Yaskawa INFORM job: SKRZYNIA_4040_-90_STOPNI_20BR.JBI

/JOB
//NAME SKRZYNIA_4040_-90_STOPNI_20BR
///FOLDERNAME 02-SKRZYNIE_JOBS
//POS
///NPOS 307,307,0,21,0,0
///TOOL 0
///POSTYPE PULSE
///PULSE
C00000=0,-52280,40443,0,6876,0
C00001=-82314,-24956,17040,-59626,-27382,-6248
C00002=-93910,-8625,17040,-59626,-43355,-6248
C00003=-98846,-1061,-42166,-80308,-57081,16120
C00004=-100452,6057,-48127,-85711,-56704,21322
C00005=-95817,31791,-34187,-84788,-63710,26674
C00006=-95573,33077,-33257,-84645,-64023,26851
C00007=-94315,33778,-32137,-85160,-63467,26714
C00008=-95573,33077,-33257,-84645,-64023,26851
C00009=-94948,31301,-36075,-85235,-63717,27152
C00010=-95573,33077,-33257,-84645,-64023,26851
C00011=-95263,33142,-33256,-84677,-63995,26850
C00012=-95263,33142,-33256,-84677,-63995,26850
C00013=-94230,33719,-32331,-85099,-63538,26735
C00014=-95263,33142,-33256,-84677,-63995,26850
C00015=-94794,31816,-35365,-85120,-63763,27076
C00016=-95263,33142,-33256,-84677,-63995,26850
C00017=-95260,33144,-33256,-84678,-63995,26850
C00018=-95260,33144,-33256,-84678,-63995,26850
C00019=-94260,33701,-32361,-85086,-63552,26738
C00020=-95738,35616,-30155,-83417,-65710,26451
C00021=-94835,31943,-35167,-85080,-63786,27056
C00022=-95260,33144,-33256,-84678,-63995,26850
C00023=-95258,25631,32269,-66559,-75499,2416
C00024=-95258,25631,32269,-66559,-75499,2416
C00025=-94256,26435,33444,-66420,-74940,2208
C00026=-95258,25631,32269,-66559,-75499,2416
C00027=-94857,24030,29962,-66606,-75105,2539
C00028=-95258,25631,32269,-66559,-75499,2416
C00029=-98811,21047,-15512,-99242,-81394,20987
C00030=-98811,21047,-15512,-99242,-81394,20987
C00031=-97856,21592,-14760,-99539,-80803,20995
C00032=-98811,21047,-15512,-99242,-81394,20987
C00033=-98487,19855,-17143,-99373,-81250,21110
C00034=-98811,21047,-15512,-99242,-81394,20987
C00035=-100395,5963,-6492,-101051,-69866,13942
C00036=-97697,-21147,-29798,-104770,-52931,14344
C00037=-81691,-45027,-49520,-104186,-37412,14105
C00038=-48287,-44591,-17414,-16172,-14532,-25809
C00039=-85348,-13130,13838,-41209,-47455,-8220
C00040=-97998,22495,32685,-69647,-75009,8900
C00041=-98284,29564,37770,-71835,-80250,10571
C00042=-100615,26523,30326,-83718,-79542,3747
C00043=-99528,26746,30653,-83688,-78804,3698
C00044=-98609,27389,31597,-83640,-78189,3601
C00045=-99528,26746,30653,-83688,-78804,3698
C00046=-99278,25562,28929,-83734,-78615,3833
C00047=-99528,26746,30653,-83688,-78804,3698
C00048=-97827,29852,38067,-72347,-79830,10157
C00049=-97362,30289,38867,-71738,-79704,10396
C00050=-96447,31020,39967,-71637,-79179,10220
C00051=-97362,30289,38867,-71738,-79704,10396
C00052=-97069,28896,36765,-71776,-79401,10550
C00053=-97362,30289,38867,-71738,-79704,10396
C00054=-99687,30516,41738,-96594,-77984,-2813
C00055=-99279,34023,49568,-96204,-78485,-4167
C00056=-98297,34881,50932,-96068,-77785,-4257
C00057=-99279,34023,49568,-96204,-78485,-4167
C00058=-98948,32155,46632,-96284,-78364,-3863
C00059=-99279,34023,49568,-96204,-78485,-4167
C00060=-100799,20404,12473,-99797,-78179,2590
C00061=-99814,-4938,-36996,-116444,-71342,12229
C00062=-82620,-30758,-83593,-142203,-62652,21635
C00063=-79591,-62427,-80212,-133576,-39445,13545
C00064=-61872,-66272,-83954,-148251,-32298,21081
C00065=-61872,-49557,-32264,-110357,-15428,1928
C00066=-71091,-37860,2722,-34648,-42002,-27792
C00067=-94097,-13222,20403,-45591,-54273,-19204
C00068=-97363,-23488,-17584,-60839,-44712,-9276
C00069=-98197,-8670,-25604,-81540,-55001,4479
C00070=-99236,18416,3235,-80713,-73731,6125
C00071=-98716,22747,8680,-80557,-75862,6048
C00072=-97982,23215,9333,-80619,-75386,5974
C00073=-98716,22747,8680,-80557,-75862,6048
C00074=-98409,21490,6932,-80649,-75627,6156
C00075=-98716,22747,8680,-80557,-75862,6048
C00076=-94729,-288,3800,-87543,-55904,1533
C00077=-77861,-26606,-19905,-76223,-21443,-3330
C00078=-46440,-50562,-32626,1826,-13880,-39178
C00079=-46440,-50562,-32626,1826,-13880,-39178
///LIMIT ON
C00080=-38692,-65390,10180,-18335,3144,1955
///LIMIT OFF
C00081=0,-52280,40443,0,6876,0
C00082=0,-52280,40443,0,6876,0
C00083=0,-43112,23163,32261,-40956,29092
C00084=-48283,-21883,28214,-25170,-26491,48363
C00085=-46664,-3144,58041,-18842,-32105,45325
C00086=-50347,-18571,12268,-49104,-16423,60029
C00087=-50509,-19000,10610,-51503,-15997,61182
C00088=-52966,-16930,12240,-56194,-17032,63176
C00089=-51879,-15912,13067,-55265,-16346,62852
C00090=-52154,-16175,12851,-55507,-16521,62938
C00091=-53227,-15612,13314,-57215,-17042,63646
C00092=-52966,-16930,12240,-56194,-17032,63176
C00093=-50703,-18403,11066,-52155,-16024,61477
C00094=-52780,-17619,11680,-55562,-17015,62889
C00095=-51306,-16241,12790,-54268,-16084,62435
C00096=-51660,-16583,12512,-54593,-16308,62551
C00097=-53327,-15718,13220,-57282,-17114,63667
C00098=-52780,-17619,11680,-55562,-17015,62889
C00099=-50704,-18401,11069,-52157,-16021,61478
C00100=-53191,-17342,11901,-56260,-17204,63181
C00101=-51773,-16022,12969,-55050,-16305,62760
C00102=-52146,-16378,12679,-55379,-16540,62876
C00103=-53214,-15820,13135,-57085,-17059,63584
C00104=-53002,-17172,12037,-56105,-17083,63128
C00105=-51005,-17995,11387,-52847,-16122,61778
C00106=-52654,-17319,11922,-55560,-16911,62904
C00107=-51372,-16113,12897,-54432,-16099,62508
C00108=-51648,-16379,12679,-54684,-16273,62598
C00109=-52952,-15703,13233,-56807,-16903,63480
C00110=-53323,-17134,12070,-56539,-17248,63304
C00111=-52826,-20105,4812,-63938,-15678,66983
C00112=-52298,-19620,5183,-63681,-15322,66914
C00113=-51076,-18450,6096,-63049,-14499,66733
C00114=-51419,-18785,5831,-63233,-14731,66786
C00115=-52680,-18133,6347,-65138,-15424,67581
C00116=-52924,-19431,7025,-60935,-16175,65505
C00117=-51752,-18759,10786,-53484,-16613,62002
C00118=-52244,-17884,11471,-54682,-16766,62529
C00119=-50303,-16031,12961,-52880,-15542,61887
C00120=-50741,-16464,12607,-53310,-15818,62044
C00121=-52416,-15612,13306,-56135,-16617,63223
C00122=-51898,-18011,11369,-54129,-16600,62301
C00123=-50945,-18019,11363,-52741,-16103,61737
C00124=-51347,-17395,11856,-53690,-16237,62152
C00125=-49990,-16073,12923,-52376,-15383,61677
C00126=-50384,-16465,12603,-52769,-15629,61822
C00127=-52066,-15616,13298,-55654,-16423,63028
C00128=-51792,-17610,11685,-54205,-16494,62350
C00129=-50945,-18019,11363,-52741,-16103,61737
C00130=-50845,-17493,11778,-52895,-15987,61824
C00131=-49521,-16191,12826,-51571,-15155,61341
C00132=-49894,-16567,12520,-51958,-15389,61484
C00133=-51728,-15654,13268,-55171,-16246,62832
C00134=-51082,-17431,11827,-53280,-16102,61986
C00135=-50028,-23690,-6096,-22921,-31075,54538
C00136=-50346,-22995,-5584,-23393,-31002,54768
C00137=-48843,-21430,-4410,-21901,-30270,54078
C00138=-49178,-21788,-4683,-22239,-30433,54235
C00139=-50538,-21100,-4158,-23908,-30654,55032
C00140=-50252,-22811,-5450,-23315,-30936,54734
C00141=-49763,-24818,-32918,-23163,-28604,59699
C00142=-49144,-24298,-32242,-22455,-28505,59304
C00143=-47766,-22458,-30816,-21237,-27774,58615
C00144=-48099,-22913,-31171,-21534,-27949,58786
C00145=-49602,-21997,-30448,-23301,-28174,59772
C00146=-49259,-23869,-32392,-22880,-28141,59533
C00147=-50713,-12366,-58367,-41124,-17813,74400
C00148=-50097,-11438,-57505,-40749,-17495,74109
C00149=-49105,-9842,-55994,-40096,-16991,73614
C00150=-49355,-10250,-56383,-40269,-17116,73742
C00151=-50506,-9357,-55529,-41571,-17503,74586
C00152=-49771,-10920,-57018,-40545,-17327,73951
C00153=-46548,-30139,-39639,-20061,-27197,57955
C00154=-48797,-26670,-6576,-20404,-32539,53259
C00155=-45389,-28224,4312,-35967,-15579,54278
C00156=-40154,-51179,-915,-24203,-8234,36524
C00157=0,-52280,40443,0,6876,0
C00158=0,-52280,40443,0,6876,0
C00159=5366,-38499,37552,-33963,-10211,16191
C00160=0,-52280,40443,0,6876,0
C00161=-82314,-24956,17040,-59626,-27382,-6248
C00162=-93910,-8625,17040,-59626,-43355,-6248
C00163=-98846,-1061,-42166,-80308,-57081,16120
C00164=-100452,6057,-48127,-85711,-56704,21322
C00165=-95564,34698,-34234,-85516,-63941,27819
C00166=-94021,36658,-30981,-84167,-64832,27454
C00167=-93851,36773,-30815,-84181,-64812,27439
C00168=-95564,34698,-34234,-85516,-63941,27819
C00169=-96930,32282,-32252,-82595,-65816,26305
C00170=-93901,32995,-31122,-83953,-64436,26132
C00171=-93891,32978,-31150,-83961,-64431,26134
C00172=-96930,32282,-32252,-82595,-65816,26305
C00173=-97719,-4194,-31542,-76086,-54596,10626
C00174=-88377,-34186,-45291,-67238,-52212,2442
C00175=-73560,-62084,7826,-28695,-34737,-3666
C00176=0,-36700,24612,42871,-31823,33862
C00177=-44403,-30110,7154,-24155,-23805,45557
C00178=-51570,-19542,10947,-41619,-21811,53396
C00179=-51570,-17239,16856,-38066,-23574,51584
C00180=-55052,-13712,19754,-43494,-24529,53873
C00181=-55307,-12713,21787,-42848,-25102,53500
C00182=-40431,-28773,9158,-17648,-23273,42875
C00183=0,-36700,24612,42871,-31823,33862
C00184=0,-52280,40443,0,6876,0
C00185=0,-52280,40443,0,6876,0
C00186=-73560,-62084,7826,-28695,-34737,-3666
C00187=-88377,-34186,-45291,-67238,-52212,2442
C00188=-99860,-8392,-35780,-75647,-56000,10650
C00189=-100432,21324,12575,-83706,-77956,7498
C00190=-100432,21324,12575,-83706,-77956,7498
C00191=-97477,24790,17443,-83584,-77881,7143
C00192=-97548,25214,18044,-83537,-78171,7107
C00193=-100432,21324,12575,-83706,-77956,7498
C00194=-100473,21504,12824,-83696,-77986,7482
C00195=-97708,25565,18549,-83502,-78342,7077
C00196=-97720,26100,19317,-83456,-78605,7025
C00197=-100432,21324,12575,-83706,-77956,7498
C00198=-99336,18440,8642,-84276,-74234,7647
C00199=-97907,25479,18429,-83510,-78268,7080
C00200=-97774,25771,18838,-83486,-78362,7054
C00201=-99336,18440,8642,-84276,-74234,7647
C00202=-88887,-29565,-44699,-91336,-36715,8429
C00203=-85230,-48302,-58733,-86716,-36654,5475
C00204=-60204,-59872,-73451,-117647,-17639,18840
C00205=-57189,-26834,-7130,-38780,-31731,51561
C00206=-55949,-20676,-3191,-39588,-29733,52121
C00207=-55884,-28531,-46032,-64057,-20842,63703
C00208=-57189,-26834,-7130,-38780,-31731,51561
C00209=-41180,-61187,4729,-17280,-8498,23442
C00210=0,-52280,40443,0,6876,0
C00211=0,-52280,40443,0,6876,0
C00212=-43180,-50572,-20637,-6552,-29302,-38834
C00213=-79425,-37128,-15462,-51820,-35721,-18807
C00214=-93702,-21743,-5664,-65079,-41536,-12324
C00215=-95468,-3718,3432,-57810,-54196,-8058
C00216=-98195,18244,29331,-65465,-72367,-4307
C00217=-96728,36447,56610,-70336,-82085,-4645
C00218=-96821,31985,42520,-71106,-80277,-1800
C00219=-99571,23446,29328,-71481,-76214,-993
C00220=-98368,-15155,-15320,-68503,-52006,-4003
C00221=-90196,-30440,-22000,-63685,-45526,-9297
C00222=-44920,-50063,-20090,-8739,-29356,-37564
C00223=-50917,-40459,4132,-34421,-18173,42391
C00224=-54964,-26842,8528,-44141,-23181,52038
C00225=-51719,-20944,8196,-48593,-18539,54728
C00226=-53338,-16066,12564,-52314,-18938,56375
C00227=-53668,-14237,17353,-48629,-20286,54493
C00228=-18010,-41727,-5437,24633,-20435,23511
C00229=-41180,-61187,4729,-17280,-8498,23442
C00230=0,-52280,40443,0,6876,0
C00231=0,-52280,40443,0,6876,0
///LIMIT ON
C00232=-37721,-67612,11381,-1325,-438,-7850
///LIMIT OFF
C00233=-43180,-50572,-20637,-6552,-29302,-38834
C00234=-79425,-37128,-15462,-51820,-35721,-18807
C00235=-92377,-33385,-41303,-83059,-36844,-1354
C00236=-98043,-4314,-16897,-86107,-58749,2387
C00237=-99186,-1007,-13605,-90357,-63007,3800
C00238=-99448,23410,16807,-87478,-77479,2357
C00239=-98529,24761,18725,-87324,-78429,2215
C00240=-98419,25196,20150,-87169,-78534,1864
C00241=-99450,-173,-12700,-90327,-63185,3798
C00242=-99875,3426,-9244,-98609,-66692,6315
C00243=-99431,-3293,-16601,-99643,-62713,6757
C00244=-92822,-26306,-37175,-103295,-43881,7703
C00245=-68601,-52593,-52127,-95725,-25602,3235
C00246=-80632,-38079,-20908,-64053,-45216,-12949
C00247=-50917,-40459,4132,-34421,-18173,42391
C00248=-51059,-36587,4608,-36647,-19418,45358
C00249=-50113,-22729,10834,-36393,-23396,50963
C00250=-58003,-17258,7975,-66354,-22196,69294
C00251=-57716,-15816,11809,-61896,-22664,66720
C00252=-50113,-22729,10834,-36393,-23396,50963
C00253=-45969,-44671,-42317,80322,10570,10889
C00254=-43180,-50572,-20637,-6552,-29302,-38834
C00255=-79425,-37128,-15462,-51820,-35721,-18807
C00256=-92377,-33385,-41303,-83059,-36844,-1354
C00257=-97955,-4566,-17156,-86109,-58691,2381
C00258=-98763,-4191,-27333,-97091,-62203,7437
C00259=-100541,17285,32324,-96596,-68502,-4435
C00260=-99163,31411,54049,-96228,-73919,-6997
C00261=-97653,31369,46884,-97568,-75920,-4787
C00262=-97653,34871,57346,-96543,-75121,-6929
C00263=-98792,6748,2422,-99606,-66785,1957
C00264=-98813,-5502,-22210,-93134,-60245,5727
C00265=-97559,-25159,-36085,-93407,-46496,3918
C00266=-68601,-52593,-52127,-95725,-25602,3235
C00267=-80632,-38079,-20908,-64053,-45216,-12949
C00268=-43180,-50572,-20637,-6552,-29302,-38834
///LIMIT ON
C00269=-37721,-67612,11381,-1325,-438,-7850
///LIMIT OFF
C00270=-44101,-76445,-48847,-15697,-17168,40457
C00271=-48984,-30078,-36716,-21434,-29637,58750
C00272=-50484,-13386,-55713,-36158,-19724,71897
C00273=-50484,-10141,-52609,-36672,-19476,72159
C00274=-57834,15023,-57436,-77444,-21310,89314
C00275=-50484,-13386,-55713,-36158,-19724,71897
C00276=-49763,-25421,-36239,-24565,-26935,60445
C00277=-50529,-22709,-3778,-22940,-31995,54502
C00278=-45389,-28224,4312,-35967,-15579,54278
C00279=-40154,-51179,-915,-24203,-8234,36524
C00280=0,-52280,40443,0,6876,0
C00281=0,-52280,40443,0,6876,0
///LIMIT ON
C00282=-37721,-67612,11381,-1325,-438,-7850
///LIMIT OFF
C00283=-43180,-50572,-20637,-6552,-29302,-38834
C00284=-43180,-50572,-20637,-6552,-29302,-38834
C00285=-91571,-17240,10754,-52986,-45776,-17944
C00286=-85565,-2479,24798,-50710,-47830,-17652
C00287=-96886,22779,17134,-75074,-74614,-730
C00288=-96886,21697,9827,-76119,-73731,1247
C00289=-99355,23812,23162,-76774,-76908,-1703
C00290=-89794,-9992,-7341,-81590,-44258,-3681
C00291=-98228,-14972,-11291,-81392,-49231,-4002
C00292=-98228,-7428,13566,-72439,-51372,-10695
C00293=-68865,-35989,-5252,-49829,-38105,-21179
C00294=-40763,-44623,-7750,-16844,-36810,-34738
C00295=10261,-46634,14475,-36899,-22136,31570
///LIMIT ON
C00296=22834,-59963,22946,-6692,-2150,9612
///LIMIT OFF
C00297=0,-52280,40443,0,6876,0
///LIMIT ON
C00298=-23708,-46776,23536,-16027,-4787,19738
///LIMIT OFF
C00299=-50917,-40459,4132,-34421,-18173,42391
C00300=-49876,-21948,7530,-68838,-10324,59148
C00301=-46721,-18942,9765,-68167,-8197,59205
C00302=-47803,-15007,12036,-78506,-8519,63985
C00303=-48173,-14749,12492,-78097,-8776,63748
C00304=-42573,-24036,4541,-56448,-5917,54155
C00305=-31287,-69981,-10850,-7253,-6843,20996
C00306=0,-52280,40443,0,6876,0
BC00000=363722
BC00001=352964
BC00002=352964
BC00003=437444
BC00004=455875
BC00005=375013
BC00006=376061
BC00007=376061
BC00008=376061
BC00009=376061
BC00010=376061
BC00011=422255
BC00012=422255
BC00013=422255
BC00014=422255
BC00015=422255
BC00016=422255
BC00017=468422
BC00018=468422
BC00019=468422
BC00020=468422
BC00021=468422
BC00022=468422
BC00023=444238
BC00024=444238
BC00025=444238
BC00026=444238
BC00027=444238
BC00028=444238
BC00029=490292
BC00030=490292
BC00031=490292
BC00032=490292
BC00033=490292
BC00034=490292
BC00035=461916
BC00036=458522
BC00037=448514
BC00038=606955
BC00039=621951
BC00040=680325
BC00041=678232
BC00042=575839
BC00043=575839
BC00044=575839
BC00045=575839
BC00046=575839
BC00047=575839
BC00048=673458
BC00049=678232
BC00050=678232
BC00051=678232
BC00052=678232
BC00053=678232
BC00054=702900
BC00055=702900
BC00056=702900
BC00057=702900
BC00058=702900
BC00059=702900
BC00060=708094
BC00061=715248
BC00062=737075
BC00063=739717
BC00064=780078
BC00065=780078
BC00066=808755
BC00067=805735
BC00068=830015
BC00069=823094
BC00070=814601
BC00071=807810
BC00072=807810
BC00073=807810
BC00074=807810
BC00075=807810
BC00076=769391
BC00077=799668
BC00078=803254
BC00079=782390
BC00080=707163
BC00081=658186
BC00082=658184
BC00083=658186
BC00084=766092
BC00085=766092
BC00086=795394
BC00087=795890
BC00088=795890
BC00089=795890
BC00090=795890
BC00091=795890
BC00092=795890
BC00093=738548
BC00094=738548
BC00095=738548
BC00096=738548
BC00097=738548
BC00098=738548
BC00099=672663
BC00100=672663
BC00101=672663
BC00102=672663
BC00103=672663
BC00104=672663
BC00105=615008
BC00106=615008
BC00107=615008
BC00108=615008
BC00109=615008
BC00110=615008
BC00111=549905
BC00112=549905
BC00113=549905
BC00114=549905
BC00115=549905
BC00116=549905
BC00117=492580
BC00118=492580
BC00119=492580
BC00120=492580
BC00121=492580
BC00122=492580
BC00123=427066
BC00124=427066
BC00125=427066
BC00126=427066
BC00127=427066
BC00128=427066
BC00129=369647
BC00130=369647
BC00131=369647
BC00132=369647
BC00133=369647
BC00134=369647
BC00135=367378
BC00136=367378
BC00137=367378
BC00138=367378
BC00139=367378
BC00140=367378
BC00141=367378
BC00142=367378
BC00143=367378
BC00144=367378
BC00145=367378
BC00146=367378
BC00147=367378
BC00148=367378
BC00149=367378
BC00150=367378
BC00151=367378
BC00152=367378
BC00153=367378
BC00154=367378
BC00155=367374
BC00156=441050
BC00157=441050
BC00158=399984
BC00159=624042
BC00160=366330
BC00161=352964
BC00162=352964
BC00163=352964
BC00164=352964
BC00165=383772
BC00166=383751
BC00167=376148
BC00168=383772
BC00169=423163
BC00170=423163
BC00171=416135
BC00172=423163
BC00173=450041
BC00174=450041
BC00175=450041
BC00176=490644
BC00177=563016
BC00178=622362
BC00179=620614
BC00180=620614
BC00181=681206
BC00182=681587
BC00183=490644
BC00184=448758
BC00185=450041
BC00186=450041
BC00187=450041
BC00188=498778
BC00189=451598
BC00190=367111
BC00191=367111
BC00192=359499
BC00193=367111
BC00194=428582
BC00195=428582
BC00196=436129
BC00197=428582
BC00198=474694
BC00199=474700
BC00200=480831
BC00201=474694
BC00202=488516
BC00203=507726
BC00204=540993
BC00205=359905
BC00206=360245
BC00207=335989
BC00208=359905
BC00209=431999
BC00210=431999
BC00211=640937
BC00212=640937
BC00213=553973
BC00214=553967
BC00215=592346
BC00216=590816
BC00217=590816
BC00218=590816
BC00219=590816
BC00220=590070
BC00221=595538
BC00222=606406
BC00223=449627
BC00224=488588
BC00225=497390
BC00226=497267
BC00227=555184
BC00228=557128
BC00229=468922
BC00230=455634
BC00231=640937
BC00232=640937
BC00233=640937
BC00234=640937
BC00235=640937
BC00236=640937
BC00237=648365
BC00238=648365
BC00239=648365
BC00240=653387
BC00241=648365
BC00242=658303
BC00243=658303
BC00244=658303
BC00245=658303
BC00246=691207
BC00247=698935
BC00248=710701
BC00249=744351
BC00250=744351
BC00251=802580
BC00252=744351
BC00253=705860
BC00254=640937
BC00255=640937
BC00256=640937
BC00257=640937
BC00258=723517
BC00259=685623
BC00260=685623
BC00261=692821
BC00262=692821
BC00263=696743
BC00264=718930
BC00265=712189
BC00266=658303
BC00267=691207
BC00268=703131
BC00269=640937
BC00270=436090
BC00271=367378
BC00272=367378
BC00273=367380
BC00274=367378
BC00275=367378
BC00276=367378
BC00277=367378
BC00278=367374
BC00279=441050
BC00280=441050
BC00281=640937
BC00282=640937
BC00283=762421
BC00284=794688
BC00285=793103
BC00286=793103
BC00287=815706
BC00288=815706
BC00289=815706
BC00290=819804
BC00291=814580
BC00292=791801
BC00293=821754
BC00294=771366
BC00295=662718
BC00296=580559
BC00297=580559
BC00298=470174
BC00299=360196
BC00300=360196
BC00301=360196
BC00302=360796
BC00303=420704
BC00304=419720
BC00305=650116
BC00306=650116
///POSTYPE BASE
///RECTAN
///RCONF 1,0,0,0,0,0,0,0,0,0,0,0,0,0,0,0,0,0,0,0,0,0,0,0
P00006=0.000,0.000,0.000,0.0000,0.0000,0.0000
P00300=-0.036,-1.505,2.318,0.0000,0.0000,0.0000
P00301=0.046,-2.112,7.779,0.0000,0.0000,0.0000
P00302=-0.180,-2.409,6.326,0.0000,0.0000,0.0000
///RCONF 0,0,0,0,0,0,0,0,0,0,0,0,0,0,0,0,0,0,0,0,0,0,0,0
P00303=-0.004,-1.437,-4.584,0.0000,0.0000,0.0000
P00304=0.028,-1.666,-4.234,0.0000,0.0000,0.0000
P00306=0.015,-2.252,-3.054,0.0000,0.0000,0.0000
P00307=0.019,-2.151,-5.077,0.0000,0.0000,0.0000
P00308=-0.003,-2.092,-4.888,0.0000,0.0000,0.0000
P00310=-0.006,-2.490,-5.925,0.0000,0.0000,0.0000
P00351=13.563,-0.027,-0.653,0.0000,0.0000,0.0000
P00352=13.252,-0.027,-0.827,0.0000,0.0000,0.0000
P00353=10.971,-0.082,0.776,0.0000,0.0000,0.0000
P00354=-0.024,2.508,-1.824,0.0000,0.0000,0.0000
P00355=-0.001,2.528,-1.131,0.0000,0.0000,0.0000
P00356=-0.034,2.921,-0.262,0.0000,0.0000,0.0000
P00357=0.003,3.386,-0.091,0.0000,0.0000,0.0000
P00358=0.014,3.037,-0.020,0.0000,0.0000,0.0000
P00359=-0.005,2.731,0.912,0.0000,0.0000,0.0000
P00360=-0.011,3.412,0.438,0.0000,0.0000,0.0000
P00361=0.018,3.050,1.253,0.0000,0.0000,0.0000
//INST
///DATE 2025/03/28 12:58
///ATTR SC,RW
///GROUP1 RB1,BS1
NOP
CALL JOB:MOVE_INTO_TUNNEL
MOVJ C00000 BC00000 VJ=30.00
MOVJ C00001 BC00001 VJ=30.00
MOVJ C00002 BC00002 VJ=30.00
MOVL C00003 BC00003 V=500.0
MOVJ C00004 BC00004 VJ=20.00
COMM '------------------------
COMM 'W65.3
COMM '------------------------
COMM MOVL C00005 BC00005 V=333.3
COMM MOVL C00006 BC00006 V=166.7 PL=0
COMM REFP 3 C00007 BC00007
COMM CALL JOB:SEARCH-R1
COMM SET P0300 P0006
COMM SFTON P0300
COMM MOVL C00008 BC00008 V=66.7 PL=0
COMM REFP 3 C00009 BC00009
COMM CALL JOB:SEARCH-R1
COMM SET P0300 P0006
COMM SFTON P0300
COMM MOVL C00010 BC00010 V=66.7 PL=0
COMM SFTOF
COMM '------------------------
COMM 'W65.5
COMM '------------------------
COMM MOVL C00011 BC00011 V=500.0
COMM MOVL C00012 BC00012 V=166.7 PL=0
COMM REFP 3 C00013 BC00013
COMM CALL JOB:SEARCH-R1
COMM SET P0301 P0006
COMM SFTON P0301
COMM MOVL C00014 BC00014 V=166.7 PL=0
COMM REFP 3 C00015 BC00015
COMM CALL JOB:SEARCH-R1
COMM SET P0301 P0006
COMM SFTON P0301
COMM MOVL C00016 BC00016 V=166.7 PL=0
COMM SFTOF
'------------------------
'W65.7
'------------------------
MOVL C00017 BC00017 V=500.0
MOVL C00018 BC00018 V=166.7 PL=0
REFP 3 C00019 BC00019
CALL JOB:SEARCH-R1
SET P0302 P0006
SFTON P0302
MOVL C00020 BC00020 V=166.7 PL=0
REFP 3 C00021 BC00021
CALL JOB:SEARCH-R1
SET P0302 P0006
SFTON P0302
MOVL C00022 BC00022 V=166.7 PL=0
SFTOF
'------------------------
'W65.10
'------------------------
MOVL C00023 BC00023 V=500.0
MOVL C00024 BC00024 V=166.7 PL=0
REFP 3 C00025 BC00025
CALL JOB:SEARCH-R1
SET P0303 P0006
SFTON P0303
MOVL C00026 BC00026 V=166.7 PL=0
REFP 3 C00027 BC00027
CALL JOB:SEARCH-R1
SET P0303 P0006
SFTON P0303
MOVL C00028 BC00028 V=166.7 PL=0
SFTOF
'------------------------
'W65.12
'------------------------
MOVL C00029 BC00029 V=500.0
MOVL C00030 BC00030 V=166.7 PL=0
REFP 3 C00031 BC00031
CALL JOB:SEARCH-R1
SET P0304 P0006
SFTON P0304
MOVL C00032 BC00032 V=166.7 PL=0
REFP 3 C00033 BC00033
CALL JOB:SEARCH-R1
SET P0304 P0006
SFTON P0304
MOVL C00034 BC00034 V=166.7 PL=0
SFTOF
'------------------------
'W65.15
'------------------------
MOVL C00035 BC00035 V=333.3
MOVL C00036 BC00036 V=500.0
MOVL C00037 BC00037 V=500.0
MOVJ C00038 BC00038 VJ=50.00
MOVL C00039 BC00039 V=500.0
MOVL C00040 BC00040 V=500.0
'------------------------
'W65.20
'------------------------
MOVL C00041 BC00041 V=166.7
MOVL C00042 BC00042 V=416.7
MOVL C00043 BC00043 V=166.7 PL=0
REFP 3 C00044 BC00044
CALL JOB:SEARCH-R1
SET P0306 P0006
SFTON P0306
MOVL C00045 BC00045 V=166.7 PL=0
REFP 3 C00046 BC00046
CALL JOB:SEARCH-R1
SET P0306 P0006
SFTON P0306
MOVL C00047 BC00047 V=166.7 PL=0
SFTOF
MOVL C00048 BC00048 V=416.7
MOVL C00049 BC00049 V=166.7 PL=0
REFP 3 C00050 BC00050
CALL JOB:SEARCH-R1
SET P0307 P0006
SFTON P0307
MOVL C00051 BC00051 V=166.7 PL=0
REFP 3 C00052 BC00052
CALL JOB:SEARCH-R1
SET P0307 P0006
SFTON P0307
MOVL C00053 BC00053 V=166.7 PL=0
SFTOF
'------------------------
'W65.23
'------------------------
MOVL C00054 BC00054 V=333.3
MOVL C00055 BC00055 V=166.7 PL=0
REFP 3 C00056 BC00056
CALL JOB:SEARCH-R1
SET P0308 P0006
SFTON P0308
MOVL C00057 BC00057 V=166.7 PL=0
REFP 3 C00058 BC00058
CALL JOB:SEARCH-R1
SET P0308 P0006
SFTON P0308
MOVL C00059 BC00059 V=166.7 PL=0
SFTOF
'------------------------
'W65.25
'------------------------
MOVL C00060 BC00060 V=666.7
MOVL C00061 BC00061 V=666.7
MOVL C00062 BC00062 V=666.7
MOVL C00063 BC00063 V=666.7
MOVL C00064 BC00064 V=666.7
MOVL C00065 BC00065 V=666.7
MOVL C00066 BC00066 V=666.7
MOVL C00067 BC00067 V=666.7
MOVL C00068 BC00068 V=666.7
MOVL C00069 BC00069 V=500.0
MOVL C00070 BC00070 V=333.3
'------------------------
'W65.28
'------------------------
MOVL C00071 BC00071 V=166.7 PL=0
REFP 3 C00072 BC00072
CALL JOB:SEARCH-R1
SET P0310 P0006
SFTON P0310
MOVL C00073 BC00073 V=166.7 PL=0
REFP 3 C00074 BC00074
CALL JOB:SEARCH-R1
SET P0310 P0006
SFTON P0310
MOVL C00075 BC00075 V=166.7 PL=0
SFTOF
'------------------------
MOVL C00076 BC00076 V=333.3
MOVL C00077 BC00077 V=333.3
MOVL C00078 BC00078 V=333.3
MOVL C00079 BC00079 V=666.7
MOVJ C00080 BC00080 VJ=50.00
MOVJ C00081 BC00081 VJ=50.00
MOVJ C00082 BC00082 VJ=10.00
MOVJ C00083 BC00083 VJ=50.00
MOVJ C00084 BC00084 VJ=30.00
MOVJ C00085 BC00085 VJ=30.00
MOVL C00086 BC00086 V=333.3
SFTOF
'------------------------
'W254A P
'------------------------
MOVJ C00087 BC00087 VJ=40.00
MOVL C00088 BC00088 V=166.7 PL=0
REFP 3 C00089 BC00089
CALL JOB:SEARCH-R1
SET P0351 P0006
SFTON P0351
MOVL C00090 BC00090 V=166.7 PL=0
REFP 3 C00091 BC00091
CALL JOB:SEARCH-R1
SET P0351 P0006
SFTON P0351
MOVL C00092 BC00092 V=166.7 PL=0
SFTOF
'------------------------
'W254A L
'------------------------
MOVJ C00093 BC00093 VJ=40.00
MOVL C00094 BC00094 V=166.7 PL=0
REFP 3 C00095 BC00095
CALL JOB:SEARCH-R1
SET P0352 P0006
SFTON P0352
MOVL C00096 BC00096 V=166.7 PL=0
REFP 3 C00097 BC00097
CALL JOB:SEARCH-R1
SET P0352 P0006
SFTON P0352
MOVL C00098 BC00098 V=166.7 PL=0
SFTOF
'------------------------
'W250A P
'------------------------
MOVJ C00099 BC00099 VJ=40.00
MOVL C00100 BC00100 V=166.7 PL=0
REFP 3 C00101 BC00101
CALL JOB:SEARCH-R1
SET P0353 P0006
SFTON P0353
MOVL C00102 BC00102 V=66.7 PL=0
REFP 3 C00103 BC00103
CALL JOB:SEARCH-R1
SET P0353 P0006
SFTON P0353
MOVL C00104 BC00104 V=66.7 PL=0
SFTOF
'------------------------
'W250A L
'------------------------
MOVJ C00105 BC00105 VJ=40.00
MOVL C00106 BC00106 V=166.7 PL=0
REFP 3 C00107 BC00107
CALL JOB:SEARCH-R1
SET P0354 P0006
SFTON P0354
MOVL C00108 BC00108 V=66.7 PL=0
REFP 3 C00109 BC00109
CALL JOB:SEARCH-R1
SET P0354 P0006
SFTON P0354
MOVL C00110 BC00110 V=166.7 PL=0
SFTOF
'------------------------
'W253A P
'------------------------
MOVJ C00111 BC00111 VJ=40.00
MOVL C00112 BC00112 V=166.7 PL=0
REFP 3 C00113 BC00113
CALL JOB:SEARCH-R1
SET P0355 P0006
SFTON P0355
MOVL C00114 BC00114 V=166.7 PL=0
REFP 3 C00115 BC00115
CALL JOB:SEARCH-R1
SET P0355 P0006
SFTON P0355
MOVL C00116 BC00116 V=166.7 PL=0
SFTOF
'------------------------
'W253A L
'------------------------
MOVJ C00117 BC00117 VJ=40.00
MOVL C00118 BC00118 V=166.7 PL=0
REFP 3 C00119 BC00119
CALL JOB:SEARCH-R1
SET P0356 P0006
SFTON P0356
MOVL C00120 BC00120 V=166.7 PL=0
REFP 3 C00121 BC00121
CALL JOB:SEARCH-R1
SET P0356 P0006
SFTON P0356
MOVL C00122 BC00122 V=166.7 PL=0
SFTOF
'------------------------
'W256A P
'------------------------
MOVJ C00123 BC00123 VJ=40.00
MOVL C00124 BC00124 V=166.7 PL=0
REFP 3 C00125 BC00125
CALL JOB:SEARCH-R1
SET P0357 P0006
SFTON P0357
MOVL C00126 BC00126 V=166.7 PL=0
REFP 3 C00127 BC00127
CALL JOB:SEARCH-R1
SET P0357 P0006
SFTON P0357
MOVL C00128 BC00128 V=166.7 PL=0
SFTOF
'------------------------
'W256A L
'------------------------
MOVJ C00129 BC00129 VJ=40.00
MOVL C00130 BC00130 V=166.7 PL=0
REFP 3 C00131 BC00131
CALL JOB:SEARCH-R1
SET P0358 P0006
SFTON P0358
MOVL C00132 BC00132 V=166.7 PL=0
REFP 3 C00133 BC00133
CALL JOB:SEARCH-R1
SET P0358 P0006
SFTON P0358
MOVL C00134 BC00134 V=166.7 PL=0
SFTOF
'------------------------
'W252A P
'------------------------
MOVL C00135 BC00135 V=666.7
MOVL C00136 BC00136 V=166.7 PL=0
REFP 3 C00137 BC00137
CALL JOB:SEARCH-R1
SET P0359 P0006
SFTON P0359
MOVL C00138 BC00138 V=166.7 PL=0
REFP 3 C00139 BC00139
CALL JOB:SEARCH-R1
SET P0359 P0006
SFTON P0359
MOVL C00140 BC00140 V=166.7 PL=0
SFTOF
'------------------------
'W252A L
'------------------------
MOVL C00141 BC00141 V=500.0
MOVL C00142 BC00142 V=166.7 PL=0
REFP 3 C00143 BC00143
CALL JOB:SEARCH-R1
SET P0360 P0006
SFTON P0360
MOVL C00144 BC00144 V=166.7 PL=0
REFP 3 C00145 BC00145
CALL JOB:SEARCH-R1
SET P0360 P0006
SFTON P0360
MOVL C00146 BC00146 V=166.7 PL=0
SFTOF
COMM '------------------------
COMM 'W255A
COMM '------------------------
COMM MOVL C00147 BC00147 V=500.0
COMM MOVL C00148 BC00148 V=166.7 PL=0
COMM REFP 3 C00149 BC00149
COMM CALL JOB:SEARCH-R1
COMM SET P0361 P0006
COMM SFTON P0361
COMM MOVL C00150 BC00150 V=166.7 PL=0
COMM REFP 3 C00151 BC00151
COMM CALL JOB:SEARCH-R1
COMM SET P0361 P0006
COMM SFTON P0361
COMM MOVL C00152 BC00152 V=166.7 PL=0
COMM SFTOF
MOVL C00153 BC00153 V=666.7
MOVL C00154 BC00154 V=666.7
MOVL C00155 BC00155 V=666.7
MOVJ C00156 BC00156 VJ=40.00
MOVJ C00157 BC00157 VJ=40.00
MOVJ C00158 BC00158 VJ=40.00
MOVJ C00159 BC00159 VJ=50.00
CALL JOB:FRONT_SEARCH_-90ST-2_4040
MOVJ C00160 BC00160 VJ=60.00
COMM MOVJ C00161 BC00161 VJ=50.00
COMM MOVJ C00162 BC00162 VJ=50.00
COMM MOVL C00163 BC00163 V=666.7
COMM MOVJ C00164 BC00164 VJ=30.00
COMM '------------------------
COMM 'W65.3
COMM '------------------------
COMM SFTON P0300
COMM MOVL C00165 BC00165 V=333.3
COMM MOVL C00166 BC00166 V=166.7 PL=0
COMM MACRO1 MJ#(0) ARGF30
COMM ARCON
COMM MOVL C00167 BC00167 V=11.7
COMM ARCOF
COMM MOVL C00168 BC00168 V=166.7
COMM SFTOF
COMM '------------------------
COMM 'W65.5
COMM '------------------------
COMM SFTON P0301
COMM MOVL C00169 BC00169 V=666.7
COMM MOVL C00170 BC00170 V=166.7 PL=0
COMM MACRO1 MJ#(0) ARGF29
COMM ARCON
COMM MOVL C00171 BC00171 V=11.7
COMM ARCOF
COMM MOVL C00172 BC00172 V=166.7
COMM SFTOF
COMM MOVL C00173 BC00173 V=500.0
COMM MOVL C00174 BC00174 V=666.7
COMM MOVJ C00175 BC00175 VJ=40.00
COMM MOVJ C00176 BC00176 VJ=50.00
COMM MOVJ C00177 BC00177 VJ=50.00
MOVL C00178 BC00178 V=666.7
'------------------------
'W250A
'------------------------
SFTON P0354
MOVL C00179 BC00179 V=666.7
MOVL C00180 BC00180 V=166.7 PL=0
MACRO1 MJ#(0) ARGF29
ARCON
SFTOF
SFTON P0353
MOVL C00181 BC00181 V=12.5
ARCOF
MOVL C00182 BC00182 V=333.3
SFTOF
MOVJ C00183 BC00183 VJ=50.00
MOVJ C00184 BC00184 VJ=60.00
MOVJ C00185 BC00185 VJ=40.00
MOVJ C00186 BC00186 VJ=50.00
MOVJ C00187 BC00187 VJ=40.00
MOVJ C00188 BC00188 VJ=30.00
MOVJ C00189 BC00189 VJ=15.00
'------------------------
'W65.7
'------------------------
SFTON P0302
MOVL C00190 BC00190 V=833.3
MOVL C00191 BC00191 V=166.7 PL=0
MACRO1 MJ#(0) ARGF30
ARCON
MOVL C00192 BC00192 V=11.7
ARCOF
MOVL C00193 BC00193 V=166.7
SFTOF
'------------------------
'W65.10
'------------------------
SFTON P0303
MOVL C00194 BC00194 V=666.7
MOVL C00195 BC00195 V=166.7 PL=0
ARCON
MOVL C00196 BC00196 V=11.7
ARCOF
MOVL C00197 BC00197 V=166.7
SFTOF
'------------------------
'W65.12
'------------------------
SFTON P0304
MOVL C00198 BC00198 V=333.3
MOVL C00199 BC00199 V=166.7 PL=0
MACRO1 MJ#(0) ARGF30
ARCON
MOVL C00200 BC00200 V=11.7
ARCOF
MOVL C00201 BC00201 V=166.7
SFTOF
'------------------------
'W65.15
'------------------------
MOVL C00202 BC00202 V=250.0
MOVL C00203 BC00203 V=416.7
MOVL C00204 BC00204 V=666.7
SFTON P0359
MOVL C00205 BC00205 V=666.7
MOVL C00206 BC00206 V=166.7 PL=0
MACRO1 MJ#(0) ARGF29
ARCON
SFTON P0358
MOVL C00207 BC00207 V=11.7
ARCOF
MOVL C00208 BC00208 V=250.0
SFTOF
MOVJ C00209 BC00209 VJ=50.00
MOVJ C00210 BC00210 VJ=50.00
MOVJ C00211 BC00211 VJ=60.00
MOVJ C00212 BC00212 VJ=40.00
MOVJ C00213 BC00213 VJ=30.00
MOVL C00214 BC00214 V=500.0
MOVL C00215 BC00215 V=333.3
'------------------------
'W65.17
'------------------------
MOVL C00216 BC00216 V=333.3
SFTON P0306
MOVL C00217 BC00217 V=166.7 PL=0
MACRO1 MJ#(0) ARGF30
ARCON
MOVL C00218 BC00218 V=11.7
ARCOF
MOVL C00219 BC00219 V=166.7
SFTOF
MOVL C00220 BC00220 V=333.3
MOVL C00221 BC00221 V=500.0
MOVJ C00222 BC00222 VJ=40.00
MOVJ C00223 BC00223 VJ=50.00
SFTON P0356
MOVL C00224 BC00224 V=500.0
MOVL C00225 BC00225 V=500.0
MOVL C00226 BC00226 V=166.7 PL=0
MACRO1 MJ#(0) ARGF29
ARCON
SFTOF
SFTON P0355
MOVL C00227 BC00227 V=12.5
ARCOF
MOVL C00228 BC00228 V=333.3
SFTOF
MOVJ C00229 BC00229 VJ=50.00
MOVJ C00230 BC00230 VJ=50.00
MOVJ C00231 BC00231 VJ=50.00
MOVJ C00232 BC00232 VJ=50.00
MOVJ C00233 BC00233 VJ=50.00
MOVJ C00234 BC00234 VJ=50.00
MOVJ C00235 BC00235 VJ=40.00
MOVL C00236 BC00236 V=333.3
'------------------------
'W65.20
'------------------------
SFTON P0307
MOVL C00237 BC00237 V=500.0
MOVL C00238 BC00238 V=333.3
MOVL C00239 BC00239 V=166.7 PL=0
MACRO1 MJ#(0) ARGF30
ARCON
MOVL C00240 BC00240 V=11.7
ARCOF
MOVL C00241 BC00241 V=250.0
SFTOF
MOVL C00242 BC00242 V=666.7
MOVL C00243 BC00243 V=333.3
MOVL C00244 BC00244 V=500.0
MOVL C00245 BC00245 V=500.0
MOVJ C00246 BC00246 VJ=50.00
MOVJ C00247 BC00247 VJ=50.00
SFTON P0352
MOVL C00248 BC00248 V=666.7
MOVL C00249 BC00249 V=500.0
MOVL C00250 BC00250 V=250.0 PL=0
MACRO1 MJ#(0) ARGF29
ARCON
SFTOF
SFTON P0351
MOVL C00251 BC00251 V=12.5
ARCOF
MOVL C00252 BC00252 V=333.3
MOVL C00253 BC00253 V=666.7
SFTOF
MOVJ C00254 BC00254 VJ=50.00
MOVJ C00255 BC00255 VJ=30.00
MOVJ C00256 BC00256 VJ=30.00
MOVJ C00257 BC00257 VJ=20.00
MOVL C00258 BC00258 V=666.7
'------------------------
'W65.23
'------------------------
MOVL C00259 BC00259 V=333.3
MOVL C00260 BC00260 V=166.7
SFTON P0308
MOVL C00261 BC00261 V=166.7 PL=0
MACRO1 MJ#(0) ARGF30
ARCON
MOVL C00262 BC00262 V=11.7
ARCOF
MOVL C00263 BC00263 V=250.0
SFTOF
'------------------------
'W65.25
MOVL C00264 BC00264 V=500.0
MOVL C00265 BC00265 V=666.7
MOVL C00266 BC00266 V=666.7
MOVJ C00267 BC00267 VJ=40.00
MOVJ C00268 BC00268 VJ=40.00
MOVJ C00269 BC00269 VJ=50.00
COMM MOVJ C00270 BC00270 VJ=40.00
COMM '------------------------
COMM 'W255A
COMM MOVL C00271 BC00271 V=500.0
COMM MOVL C00272 BC00272 V=666.7
COMM SFTON P0361
COMM MOVL C00273 BC00273 V=166.7 PL=0
COMM MACRO1 MJ#(0) ARGF29
COMM ARCON
COMM MOVL C00274 BC00274 V=12.5
COMM ARCOF
COMM MOVL C00275 BC00275 V=333.3
COMM SFTOF
COMM MOVL C00276 BC00276 V=666.7
COMM MOVL C00277 BC00277 V=666.7
COMM MOVL C00278 BC00278 V=666.7
COMM MOVJ C00279 BC00279 VJ=50.00
COMM MOVJ C00280 BC00280 VJ=70.00
MOVJ C00281 BC00281 VJ=70.00
MOVJ C00282 BC00282 VJ=50.00
MOVJ C00283 BC00283 VJ=50.00
MOVJ C00284 BC00284 VJ=50.00
MOVL C00285 BC00285 V=500.0
'------------------------
'W31.28
'------------------------
SFTON P0310
MOVL C00286 BC00286 V=333.3
MACRO1 MJ#(0) ARGF30
MOVL C00287 BC00287 V=200.0
ARCON
MOVL C00288 BC00288 V=11.7
ARCOF
MOVL C00289 BC00289 V=166.7
SFTOF
MOVL C00290 BC00290 V=166.7
MOVL C00291 BC00291 V=500.0
MOVL C00292 BC00292 V=500.0
MOVL C00293 BC00293 V=666.7
MOVJ C00294 BC00294 VJ=25.00
MOVJ C00295 BC00295 VJ=50.00
MOVJ C00296 BC00296 VJ=50.00
MOVJ C00297 BC00297 VJ=60.00
'------------------------
'W256A
'------------------------
MOVJ C00298 BC00298 VJ=60.00
MOVJ C00299 BC00299 VJ=60.00
SFTON P0358
MOVL C00300 BC00300 V=666.7
MOVL C00301 BC00301 V=250.0
MOVL C00302 BC00302 V=166.7 PL=0
MACRO1 MJ#(0) ARGF29
ARCON
SFTOF
SFTON P0357
MOVL C00303 BC00303 V=12.5
ARCOF
MOVL C00304 BC00304 V=333.3
SFTOF
MOVJ C00305 BC00305 VJ=50.00
MOVJ C00306 BC00306 VJ=50.00
CALL JOB:FRONT_WELD_-90ST-2_4040
CALL JOB:MOVE_OUT_OF_TUNNEL
END
